FUNCTION_BLOCK LinearPosition EXTENDS SM_LinearPosition
VAR_INPUT
END_VAR
VAR_OUTPUT
END_VAR
VAR
    _testVar_LinearPosition : INT;
END_VAR

SUPER^();

// do stuff

//SUPER^();

END_FUNCTION_BLOCK

(* stored: Version 1.1.0.1, ProductVersion 3.1.4018.2
   POU LinearPosition: Id {90c58a97-434a-4c49-b49b-b7dec7933b73}, SpecialFunc None *)
